(* CoDeSys 2.3 export: ST_LINEAR_CAL.EXP *)

(* Data type *)
TYPE ST_LINEAR_CAL :
STRUCT
	K   : REAL;
	Off : REAL;
END_STRUCT
END_TYPE
